// TwinCAT 3 PLC project Sample02
// ProgramVersion: 3.1.4020.10
// libraries:
//   Tc2_Standard, * (Beckhoff Automation GmbH)
//   Tc2_System, * (Beckhoff Automation GmbH)
//   Tc3_Module, * (Beckhoff Automation GmbH)
// project tree:
//   / PlcTask.TcTTO (not stored)
//   POUs/ Class Diagram.TcCD (not stored), FB_AnalogValue.TcPOU, FB_Controller.TcPOU (not stored), FB_Lamp.TcPOU, FB_LampSetDirectDALI.TcPOU (not stored), FB_LampOnOffAdapter.TcPOU (not stored), FB_LampSetDirectAdapter.TcPOU (not stored), FB_LampSetDirectDALIAdapter.TcPOU, FB_LampUpDown.TcPOU, FB_LampSetDirect.TcPOU (not stored), FB_LampOnOff.TcPOU (not stored), FB_LampUpDownAdapter.TcPOU (not stored), I_Lamp.TcIO (not stored), I_Observer.TcIO (not stored), I_Subject.TcIO (not stored), MAIN.TcPOU (not stored)
// real-time tasks:
//   TASK PlcTask: cycle T#10ms, priority 20, ADS port 350

// ---- POUs/FB_AnalogValue.TcPOU
FUNCTION_BLOCK PUBLIC FB_AnalogValue IMPLEMENTS I_Observer
VAR_INPUT
END_VAR
VAR_OUTPUT
END_VAR
VAR
	_nActualValue		: USINT;
END_VAR

{attribute 'monitoring' := 'call'}
PROPERTY nValue : USINT
GET
nValue := _nActualValue;
END_GET
END_PROPERTY

METHOD Update
VAR_INPUT
	nNewValue		: USINT;
END_VAR
_nActualValue := nNewValue;
END_METHOD

END_FUNCTION_BLOCK

// ---- POUs/FB_Lamp.TcPOU
FUNCTION_BLOCK PUBLIC ABSTRACT FB_Lamp IMPLEMENTS I_Subject, I_Lamp
VAR
	_ipObserver		: I_Observer;
	_bIsDALIDevice	: BOOL := FALSE;
END_VAR

METHOD PUBLIC Attach
VAR_INPUT
	ipObserver		: I_Observer;
END_VAR
IF (ipObserver = 0) THEN
	RETURN;
END_IF
_ipObserver := ipObserver;
END_METHOD

// Is TRUE, if the lamp is a DALI device.
{attribute 'monitoring' := 'call'} 
PROPERTY PUBLIC bIsDALIDevice : BOOL
GET
bIsDALIDevice := _bIsDALIDevice;
END_GET
SET
_bIsDALIDevice := bIsDALIDevice;
END_SET
END_PROPERTY

METHOD PUBLIC Detach
_ipObserver := 0;
END_METHOD

// Reduces the control value by 5 in the range of 10 to 100.
METHOD PUBLIC ABSTRACT DimDown
END_METHOD

// Increments the control value by 5 in the range of 10 to 100.
METHOD PUBLIC ABSTRACT DimUp
END_METHOD

// Sets the control value to 0.
METHOD PUBLIC ABSTRACT Off
END_METHOD

// Sets the control value to 100.
METHOD PUBLIC ABSTRACT On
END_METHOD

END_FUNCTION_BLOCK

// ---- POUs/FB_LampSetDirectDALIAdapter.TcPOU
FUNCTION_BLOCK PUBLIC FB_LampSetDirectDALIAdapter EXTENDS FB_Lamp
VAR
	fbLampSetDirectDALI		: FB_LampSetDirectDALI;
END_VAR

// Reduces the control value by 5 in the range of 10 to 254.
METHOD PUBLIC DimDown
IF (fbLampSetDirectDALI.nLightLevel >= 38.1) THEN
	fbLampSetDirectDALI.SetLightLevel(TO_BYTE(fbLampSetDirectDALI.nLightLevel - 12.7));
END_IF
IF (_ipObserver <> 0) THEN
	_ipObserver.Update(fbLampSetDirectDALI.nLightLevel);
END_IF
END_METHOD

// Increments the control value by 5 in the range of 10 to 254.
METHOD PUBLIC DimUp
IF (fbLampSetDirectDALI.nLightLevel <= 241.3) THEN
	fbLampSetDirectDALI.SetLightLevel(TO_BYTE(TO_LREAL(fbLampSetDirectDALI.nLightLevel) + 12.7));
END_IF
IF (_ipObserver <> 0) THEN
	_ipObserver.Update(fbLampSetDirectDALI.nLightLevel);
END_IF
END_METHOD

METHOD FB_init : BOOL
VAR_INPUT
	bInitRetains : BOOL; // if TRUE, the retain variables are initialized (warm start / cold start)
	bInCopyCode : BOOL;  // if TRUE, the instance afterwards gets moved into the copy code (online change)
END_VAR
SUPER^._bIsDALIDevice := TRUE;
END_METHOD

// Sets the control value to 0.
METHOD PUBLIC Off
fbLampSetDirectDALI.SetLightLevel(0);
IF (_ipObserver <> 0) THEN
	_ipObserver.Update(fbLampSetDirectDALI.nLightLevel);
END_IF
END_METHOD

// Sets the control value to 254.
METHOD PUBLIC On
fbLampSetDirectDALI.SetLightLevel(254);
IF (_ipObserver <> 0) THEN
	_ipObserver.Update(fbLampSetDirectDALI.nLightLevel);
END_IF
END_METHOD

END_FUNCTION_BLOCK

// ---- POUs/FB_LampUpDown.TcPOU
FUNCTION_BLOCK FB_LampUpDown
VAR
	nLightLevel			: USINT;
END_VAR

// Reduces the control value by 1 in the range of 10 to 100.
METHOD PUBLIC OneStepDown
nLightLevel := nLightLevel - 1;
IF (nLightLevel < 10) THEN
	nLightLevel := 10;
END_IF
END_METHOD

// Increments the control value by 1 in the range of 10 to 100.
METHOD PUBLIC OneStepUp
nLightLevel := nLightLevel + 1;
IF (nLightLevel > 100) THEN
	nLightLevel := 100;
END_IF
END_METHOD

// Toggles the control value between 0 and 100.
METHOD PUBLIC OnOff
IF (nLightLevel > 0) THEN
	nLightLevel := 0;
ELSE
	nLightLevel := 100;
END_IF
END_METHOD

END_FUNCTION_BLOCK
